(* PLC project TC3_TE1400_GeneratedModule_controller_ballcatcher_FB, Beckhoff Automation GmbH & Co. KG TwinCAT 3 Function - TE1400 1.2.1237 *)
(* stored: companyURL www.beckhoff.com, creationDateTime 2020-10-13T20:18:50 *)

TYPE E_TcMatSimDataAreaType : (NotSpecified := 0, Standard, InputSrc, InputDst, OutputSrc, OutputDst, InternalDa, MArea, RetainDa);
END_TYPE

TYPE ST_TcMatSimObjectDataAreaInfo : STRUCT
  pPlcVar : PVOID;
  pModuleProcImg : PVOID;
  nSize : UDINT;
  nDataAreaId : UDINT;
  eDataAreaType : E_TcMatSimDataAreaType;
END_STRUCT;
END_TYPE

{attribute 'pack_mode' := '4'}
TYPE ST_controller_ballcatcherInitData : STRUCT
  Header : TComInitDataHdr;
  CallByHdr : TComInitDataElmHdr;
  CallBy : TctModuleCallByType;
  ExecutionSequenceHdr : TComInitDataElmHdr;
  ExecutionSequence : TctModuleExecutionSequenceType;
  StepSizeHdr : TComInitDataElmHdr;
  StepSize : TctStepSizeType;
  ExtModeParametersHdr : TComInitDataElmHdr;
  ExtModeParameters : TctExtModeParametersType;
  ExecuteModelCodeHdr : TComInitDataElmHdr;
  ExecuteModelCode : BOOL;
  ModelParametersHdr : TComInitDataElmHdr;
  ModelParameters : P_controller_ballcatcher_T;
  ContextInfoArr_0_TaskOidHdr : TComInitDataElmHdr;
  ContextInfoArr_0_TaskOid : OTCID;
  ContextInfoArr_0_TaskPriorityHdr : TComInitDataElmHdr;
  ContextInfoArr_0_TaskPriority : UDINT;
  ContextInfoArr_0_TaskCycleTimeNsHdr : TComInitDataElmHdr;
  ContextInfoArr_0_TaskCycleTimeNs : UDINT;
  ContextInfoArr_0_TaskPortHdr : TComInitDataElmHdr;
  ContextInfoArr_0_TaskPort : UINT;
  ContextInfoArr_0_TaskSortOrderHdr : TComInitDataElmHdr;
  ContextInfoArr_0_TaskSortOrder : UDINT;
END_STRUCT;
END_TYPE

TYPE ST_controller_ballcatcher_Input : STRUCT
  fast_sensor_torque : matrix_7_real_T;
  fast_sensor_position : matrix_7_real_T;
  fast_sensor_motor_torque_feedback : matrix_7_real_T;
  motion_enabled : LREAL;
  sensor_mft_application_button : LREAL;
  q_d_in : matrix_7_real_T;
  traj_time_interval : matrix_2_real_T;
  traj_update_index : LREAL;
  traj_reset : LREAL;
  chart_state : LREAL;
  controller_select : UDINT;
END_STRUCT;
END_TYPE

TYPE ST_controller_ballcatcher_Output : STRUCT
  fast_control_motor_torque : matrix_7_real_T;
  fast_control_motor_enable : matrix_7_real_T;
  motion_enabled_out : LREAL;
  traj_gen_error : BOOL;
  q_d : matrix_7_real_T;
  q_p_d : matrix_7_real_T;
  q_pp_d : matrix_7_real_T;
END_STRUCT;
END_TYPE

FUNCTION_BLOCK FB_TcMatSimObject
  VAR_INPUT
    bWriteFbInputValues : BOOL := TRUE;  (* set this flag to write FB input values to the TcComObject's input DataAreas. This will overwrite the mapped input values before module execution. Set to FALSE to read the mapped input values from the TcComObject to the FB. *)
  END_VAR
  VAR
    pDataAreas : POINTER TO ST_TcMatSimObjectDataAreaInfo;  (* process image src and dst pointers and sizes *)
    nDataAreas : UDINT;
    ipObjSrv : ITComObjectServer;  (* global interface pointers *)
    ipTcComObj : ITComObject;  (* object interface pointers *)
    ipTcCyclic : ITcCyclic;
    ipTcPostCyclic : ITcPostCyclic;
    ipTcAdi : ITcADI;
    ipTask : ITcTask;  (* task interface pointers *)
    pInitData : POINTER TO TComInitDataHdr;  (* initial parameters *)
    hResult : HRESULT;  (* hResult of interface calls (0 if no error) *)
    moduleClsId : CLSID;  (* module class ID *)
    assignedClsId : CLSID;  (* expected/desired module class ID *)
    bClassIdVerified : BOOL;
    bDynInstance : BOOL;  (* flag indicating whether the module instance was created dynamically *)
    eInitialObjState : TCOM_STATE := TCOM_STATE.TCOM_STATE_INIT;  (* the object state at the time FB_init was called, FB_exit will try to switch to this state (only if this means to shift down) *)
  END_VAR

            
          

{attribute 'object_name' := 'ReleaseTcComInterface'}
METHOD ReleaseTcComInterface : HRESULT
  VAR
    nStateChangeCnt : DINT := 0;
  END_VAR
                  
IF (ipTcComObj<>0) THEN
  WHILE (State>eInitialObjState AND nStateChangeCnt<1000) DO
    State := eInitialObjState;
    nStateChangeCnt := nStateChangeCnt+1;
  END_WHILE
  ReleaseObjInterfaces();
  IF (bDynInstance) THEN
    ReleaseTcComInterface := TC3_MODULE.FW_ObjMgr_DeleteInstance(ADR(ipTcComObj));
  ELSE
    ipTcComObj.TcRelease();
  END_IF
  ipTcComObj := 0;
END_IF
                  
                
END_METHOD

{attribute 'object_name' := 'ReleaseObjInterfaces'}
METHOD ReleaseObjInterfaces : HRESULT
                  
// release interface pointers
IF (ipTcCyclic<>0) THEN
  ipTcCyclic.TcRelease();
  ipTcCyclic := 0;
END_IF
IF (ipTcPostCyclic<>0) THEN
  ipTcPostCyclic.TcRelease();
  ipTcPostCyclic := 0;
END_IF
IF (ipTcAdi<>0) THEN
  ipTcAdi.TcRelease();
  ipTcAdi := 0;
END_IF
                  
                
END_METHOD

{attribute 'object_name' := 'Internal_SetObjState'}
METHOD Internal_SetObjState
  VAR_INPUT
    hr : REFERENCE TO HRESULT;
    nextState : TCOM_STATE;
  END_VAR
                  
// verify class id
IF (SUCCEEDED(hr)) THEN
  hr := VerifyClassId();
END_IF

// switch object state
IF (SUCCEEDED(hr) AND nextState>=TCOM_STATE_INIT) THEN
  IF (ipTcComObj=0) THEN
    hr := Tc2_System.E_HRESULTAdsErr.NOINTERFACE;
  END_IF
  IF (ipObjSrv=0) THEN
    hr := Tc2_System.E_HRESULTAdsErr.NOINTERFACE;
  END_IF
  IF (SUCCEEDED(hr)) THEN
    hr := ipTcComObj.TcSetObjState(nextState,ipObjSrv,pInitData);
  END_IF
END_IF
                  
                
END_METHOD

{attribute 'object_name' := 'FB_init'}
METHOD FB_init : BOOL
  VAR_INPUT
    bInitRetains : BOOL;  (* init retain variables *)
    bInCopyCode : BOOL;  (* Online Change *)
    oid : OTCID;
  END_VAR
                  
FB_init := SUCCEEDED(Init(oid));
                  
                
END_METHOD

{attribute 'object_name' := 'GetObjPara'}
METHOD GetObjPara : HRESULT
  VAR_INPUT
    pid : PTCID;
    nData : UDINT;
    pData : PVOID;
  END_VAR
                  
IF (ipTcComObj=0) THEN
  GetObjPara := Tc2_System.E_HRESULTAdsErr.NOINTERFACE;
END_IF

IF (SUCCEEDED(GetObjPara)) THEN
  GetObjPara := ipTcComObj.TcGetObjPara(pid:=pid,nData,pData,0);
END_IF
                  
                
END_METHOD

{attribute 'object_name' := 'QueryObjInterface'}
METHOD QueryObjInterface
  VAR_INPUT
    hr : REFERENCE TO HRESULT;
    iid : REFERENCE TO IID;
    pipItf : POINTER TO ITcUnknown;
  END_VAR
  VAR CONSTANT
    pNull : PVOID := 0;
  END_VAR
                  
IF (SUCCEEDED(hr)) THEN
  IF (ipTcComObj=0) THEN
    hr := Tc2_System.E_HRESULTAdsErr.NOINTERFACE;
  ELSIF (pipItf^=ULINT_TO_DWORD(pNull)) THEN
    hr := ipTcComObj.TcQueryInterface(iid:= iid, pipItf:=pipItf);
  END_IF
END_IF
                  
                
END_METHOD

{attribute 'object_name' := 'SaveOnlineParametersForInit'}
METHOD SaveOnlineParametersForInit : HRESULT
  VAR
    idx : UINT;
    pInitElemHdr : POINTER TO TComInitDataElmHdr;
    pData : PVOID;
    nData : UDINT;
  END_VAR
  VAR CONSTANT
    nInitDataAlignment : UDINT := 4;
  END_VAR
                  IF (pInitData<>0) THEN
  pInitElemHdr := pInitData + SIZEOF(pInitData^);
  FOR idx:=1 TO pInitData^.uiElmCnt DO
    pData := pInitElemHdr + ULINT_TO_DWORD(SIZEOF(pInitElemHdr^));
    nData := pInitElemHdr^.cbData;
    SaveOnlineParametersForInit := GetObjPara(pInitElemHdr^.indexOffset,nData,pData);
    IF (FAILED(SaveOnlineParametersForInit)) THEN
      RETURN;
    END_IF
    pInitElemHdr := pData + (nInitDataAlignment*((nData + nInitDataAlignment - 1)/nInitDataAlignment));
  END_FOR
ELSE
	SaveOnlineParametersForInit := Tc2_System.E_HRESULTAdsErr.NOTINIT;
END_IF
                  
                
END_METHOD

{attribute 'object_name' := 'ResetHresult'}
METHOD ResetHresult
                  hResult := S_OK;
                
END_METHOD

{attribute 'object_name' := 'Execute'}
METHOD Execute : HRESULT
  VAR
    nDaIdx : UDINT;
    pCurDataArea : POINTER TO ST_TcMatSimObjectDataAreaInfo;
  END_VAR
                  
IF (SUCCEEDED(hResult)) THEN
  hResult := VerifyClassId();
END_IF

IF (SUCCEEDED(hResult) AND State<>TCOM_STATE_OP) THEN
  hResult := Tc2_System.E_HRESULTAdsErr.NOTREADY;
END_IF

// get image pointers
IF (SUCCEEDED(hResult)) THEN
  GetImagePtrs(hResult);
END_IF

// copy inputs
IF (pDataAreas<>0 AND nDataAreas>0 AND bWriteFbInputValues) THEN
  FOR nDaIdx:=0 TO nDataAreas-1 DO
    IF (FAILED(hResult))THEN
      CONTINUE;
    END_IF
    pCurDataArea := pDataAreas + nDaIdx*SIZEOF(ST_TcMatSimObjectDataAreaInfo);
    IF ((pCurDataArea^.eDataAreaType <> E_TcMatSimDataAreaType.InputDst))THEN
      CONTINUE;
    END_IF
    IF (pCurDataArea^.pModuleProcImg<>0 AND pCurDataArea^.pPlcVar<>0) THEN
      MEMCPY(pCurDataArea^.pModuleProcImg,pCurDataArea^.pPlcVar,pCurDataArea^.nSize);
    ELSE
      hResult := Tc2_System.E_HRESULTAdsErr.NOINTERFACE;
    END_IF
  END_FOR
END_IF

// call cycle update
IF (SUCCEEDED(hResult)) THEN
  IF (ipTcCyclic<>0) THEN
    hResult := ipTcCyclic.CycleUpdate(ipTask:= ipTask, ipCaller:= 0, context:= 0);
  ELSE
    hResult := Tc2_System.E_HRESULTAdsErr.NOINTERFACE;
  END_IF
END_IF

// copy outputs
IF (pDataAreas<>0 AND nDataAreas>0) THEN
  FOR nDaIdx:=0 TO nDataAreas-1 DO
    IF (FAILED(hResult))THEN
      CONTINUE;
    END_IF
    pCurDataArea := pDataAreas + nDaIdx*SIZEOF(ST_TcMatSimObjectDataAreaInfo);
    IF ((pCurDataArea^.eDataAreaType = E_TcMatSimDataAreaType.OutputSrc) OR NOT bWriteFbInputValues) THEN
      IF (pCurDataArea^.pModuleProcImg<>0 AND pCurDataArea^.pPlcVar<>0) THEN
        MEMCPY(pCurDataArea^.pPlcVar,pCurDataArea^.pModuleProcImg,pCurDataArea^.nSize);
      ELSE
        hResult := Tc2_System.E_HRESULTAdsErr.NOINTERFACE;
      END_IF
    END_IF
  END_FOR
END_IF


// call post cyclic update
IF (SUCCEEDED(hResult)) THEN
  IF (ipTcPostCyclic<>0) THEN
    hResult := ipTcPostCyclic.PostCyclicUpdate(ipTask:= 0, ipCaller:= 0, context:= 0);
  ELSE
    hResult := Tc2_System.E_HRESULTAdsErr.NOINTERFACE;
  END_IF
END_IF

ReleaseImagePtrs();

Execute := hResult;
                  
                
END_METHOD

{attribute 'object_name' := 'GetImagePtrs'}
METHOD GetImagePtrs
  VAR_INPUT
    hr : REFERENCE TO HRESULT;
  END_VAR
  VAR
    nDaIdx : UDINT;
    pCurDataArea : POINTER TO ST_TcMatSimObjectDataAreaInfo;
  END_VAR
                  
IF (ipTcAdi=0) THEN
  hr := Tc2_System.E_HRESULTAdsErr.NOINTERFACE;
END_IF
IF(State<>TCOM_STATE_OP)THEN
  hr := Tc2_System.E_HRESULTAdsErr.INVALIDSTATE;
END_IF


// get pointers to process images
IF (pDataAreas<>0 AND nDataAreas>0) THEN
  FOR nDaIdx:=0 TO nDataAreas-1 DO
    pCurDataArea := pDataAreas + nDaIdx*SIZEOF(ST_TcMatSimObjectDataAreaInfo);
    IF (FAILED(hr))THEN
      CONTINUE;
    END_IF
    IF ((pCurDataArea^.eDataAreaType <> E_TcMatSimDataAreaType.InputDst) AND (pCurDataArea^.eDataAreaType <> E_TcMatSimDataAreaType.OutputSrc))THEN
      CONTINUE;
    END_IF
    IF (pCurDataArea^.pModuleProcImg=0 AND pCurDataArea^.nSize>0) THEN
      hr := ipTcAdi.GetImagePtr(size:= pCurDataArea^.nSize , offs:=0 , adi_x:=pCurDataArea^.nDataAreaId , ppData:=ADR(pCurDataArea^.pModuleProcImg));
    END_IF
  END_FOR
END_IF

IF (FAILED(hr)) THEN
  ReleaseImagePtrs();
END_IF
                  
                
END_METHOD

{attribute 'object_name' := 'VerifyClassId'}
METHOD VerifyClassId : HRESULT
  VAR
    emptyClsId : CLSID;
  END_VAR
                  memset(ADR(emptyClsId),0,SIZEOF(emptyClsId));
IF (bClassIdVerified) THEN
  // class ID was already verified
  VerifyClassId := Tc2_System.E_HRESULTAdsErr.HRESULT_ADS_NOERROR;
ELSIF (memcmp(ADR(assignedClsId),ADR(emptyClsId),SIZEOF(assignedClsId))=0) THEN
  // skip class ID verification if no assignedClsId specified
  VerifyClassId := Tc2_System.E_HRESULTAdsErr.HRESULT_ADS_NOERROR;
ELSE
  // verify class ID
  VerifyClassId := ReadModuleClassId();

  IF (SUCCEEDED(VerifyClassId)) THEN
    IF (memcmp(ADR(assignedClsId),ADR(moduleClsId),SIZEOF(assignedClsId))<>0) THEN
     VerifyClassId := Tc2_System.E_HRESULTAdsErr.INVALIDCLSID;
    END_IF
  END_IF
  bClassIdVerified := SUCCEEDED(VerifyClassId);
END_IF
                  
                
END_METHOD

{attribute 'object_name' := 'SetObjPara'}
METHOD SetObjPara : HRESULT
  VAR_INPUT
    pid : PTCID;
    nData : UDINT;
    pData : PVOID;
  END_VAR
                  
IF (ipTcComObj=0) THEN
  SetObjPara := Tc2_System.E_HRESULTAdsErr.NOINTERFACE;
END_IF

IF (SUCCEEDED(SetObjPara)) THEN
  SetObjPara := ipTcComObj.TcSetObjPara(pid:=pid,nData,pData,0);
END_IF
                  
                
END_METHOD

{attribute 'object_name' := 'QueryTcComInterface'}
METHOD QueryTcComInterface
  VAR_INPUT
    hr : REFERENCE TO HRESULT;
    oid : OTCID;
  END_VAR
                  
IF (ipObjSrv=0) THEN
  hr := Tc2_System.E_HRESULTAdsErr.NOINTERFACE;
END_IF

IF (SUCCEEDED(hr) AND ipTcComObj=0) THEN
  bDynInstance := FALSE;
  IF(oid>0) THEN
    // query interface of existing object
    hr := ipObjSrv.TcQueryObjectInterface(oid,IID_ITComObject,ADR(ipTcComObj));
  ELSE
    // create new instance and get the object interface
    hr := ipObjSrv.TcCreateInstance(assignedClsId,IID_ITComObject,ADR(ipTcComObj));
    IF (SUCCEEDED(hr)) THEN
      bDynInstance := TRUE;
      hr := ipTcComObj.TcSetObjectId(OTCID_CreateNewId);
    END_IF
  END_IF
  IF (SUCCEEDED(hr)) THEN
    eInitialObjState := State;
  END_IF
END_IF
                  
                
END_METHOD

{attribute 'object_name' := 'ReleaseImagePtrs'}
METHOD ReleaseImagePtrs : HRESULT
  VAR
    nDaIdx : UDINT;
    pCurDataArea : POINTER TO ST_TcMatSimObjectDataAreaInfo;
  END_VAR
                  
IF (ipTcAdi=0) THEN
  ReleaseImagePtrs := Tc2_System.E_HRESULTAdsErr.NOINTERFACE;
END_IF

IF (SUCCEEDED(ReleaseImagePtrs) AND pDataAreas<>0 AND nDataAreas>0) THEN
  // release pointers to the simulink module process images
  FOR nDaIdx:=0 TO nDataAreas-1 DO
    pCurDataArea := pDataAreas + nDaIdx*SIZEOF(ST_TcMatSimObjectDataAreaInfo);

    IF (pCurDataArea^.pModuleProcImg<>0) THEN
      ipTcAdi.ReleaseImagePtr(pData:=pCurDataArea^.pModuleProcImg);
      pCurDataArea^.pModuleProcImg := 0;
    END_IF
  END_FOR
END_IF
                  
                
END_METHOD

{attribute 'object_name' := 'FB_exit'}
METHOD FB_exit : BOOL
  VAR_INPUT
    bInCopyCode : BOOL;  (* Online Change *)
  END_VAR
                  
IF (NOT bInCopyCode) THEN
  IF (ipObjSrv<>0) THEN
    ipObjSrv.TcRelease();
    ipObjSrv := 0;
  END_IF

  ReleaseTcComInterface();
END_IF
                  
                
END_METHOD

{attribute 'object_name' := 'InitObjName'}
METHOD InitObjName
  VAR_INPUT
    hr : REFERENCE TO HRESULT;
  END_VAR
  VAR
    objectName : STRING(255) := 'TcMatSimObject_PlcRtFbInstance';
    oid : OTCID;
  END_VAR
                  
IF (SUCCEEDED(hr)) THEN
  hr := ipTcComObj.TcGetObjectId(oid);
END_IF

IF (SUCCEEDED(hr) and bDynInstance) THEN
  objectName := TC2_STANDARD.CONCAT(objectName,'_');
  objectName := TC2_STANDARD.CONCAT(objectName,UDINT_TO_STRING(oid));
  hr := ipTcComObj.TcSetObjectName(ADR(objectName));
END_IF
                  
                
END_METHOD

{attribute 'object_name' := 'SetObjState'}
METHOD SetObjState : HRESULT
  VAR_INPUT
    finalState : TCOM_STATE;
  END_VAR
  VAR
    bShiftUp : BOOL;
    bShiftDown : BOOL;
    currentState : TCOM_STATE;
  END_VAR
                  
currentState := State;

bShiftUp := finalState>currentState;
bShiftDown := finalState<currentState;

// do not switch up on error
IF (FAILED(hresult)) THEN
  bShiftUp := FALSE;
END_IF
// reset existing error on switching down
IF (bShiftDown) THEN
  ResetHresult();
END_IF

// prepared state switch
CASE currentState OF
  TCOM_STATE_INIT:
    IF(bShiftUp) THEN
      QueryTcComInterface(hResult,0);
      Internal_SetObjState(hResult,TCOM_STATE.TCOM_STATE_PREOP);
      InitObjName(hResult);
    END_IF

  TCOM_STATE_PREOP:
    IF(bShiftUp) THEN
      Internal_SetObjState(hResult,TCOM_STATE.TCOM_STATE_SAFEOP);
      QueryObjInterfaces(hResult);
    ELSIF (bShiftDown) THEN
      Internal_SetObjState(hResult,TCOM_STATE.TCOM_STATE_INIT);
    END_IF

  TCOM_STATE_SAFEOP:
    IF(bShiftUp) THEN
      Internal_SetObjState(hResult,TCOM_STATE.TCOM_STATE_OP);
      QueryObjInterfaces(hResult);
    ELSIF (bShiftDown) THEN
      Internal_SetObjState(hResult,TCOM_STATE.TCOM_STATE_PREOP);
      ReleaseObjInterfaces();
    END_IF


  TCOM_STATE_OP:
    IF (bShiftDown) THEN
      Internal_SetObjState(hResult,TCOM_STATE.TCOM_STATE_SAFEOP);
    END_IF
END_CASE

SetObjState := hResult;
                  
                
END_METHOD

{attribute 'object_name' := 'QueryObjInterfaces'}
METHOD QueryObjInterfaces
  VAR_INPUT
    hr : REFERENCE TO HRESULT;
  END_VAR
                  
IF(State<TCOM_STATE_PREOP)THEN
  hr := Tc2_System.E_HRESULTAdsErr.INVALIDSTATE;
END_IF

//cyclic interface
QueryObjInterface(hr,IID_ITCCYCLIC,ADR(ipTcCyclic));
//post cyclic interface
QueryObjInterface(hr,IID_ITCPOSTCYCLIC,ADR(ipTcPostCyclic));
//adi interface
QueryObjInterface(hr,IID_ITcADI,ADR(ipTcAdi));
                  
                
END_METHOD

{attribute 'object_name' := 'Init'}
METHOD Init : HRESULT
  VAR_INPUT
    oid : OTCID;
  END_VAR
                  
// preinitialize variables
memset(ADR(moduleClsId),0,SIZEOF(moduleClsId));
bClassIdVerified := FALSE;
hResult := Tc2_System.E_HRESULTAdsErr.HRESULT_ADS_NOERROR;

// get object server
IF (ipObjSrv=0) THEN
  hResult := FW_ObjMgr_GetObjectServer(_AppInfo.ObjId,ADR(ipObjSrv));
END_IF

// try to get object interfaces
IF (SUCCEEDED(hresult)) THEN
  QueryTcComInterface(hResult,oid);
END_IF

// verify class id
IF (SUCCEEDED(hresult)) THEN
  hresult := VerifyClassId();
END_IF

// query interfaces, if the current state is higher than INIT
IF (SUCCEEDED(hresult) AND State>TCOM_STATE.TCOM_STATE_INIT) THEN
  QueryObjInterfaces(hResult);
END_IF

// return value
Init := hresult;
                  
                
END_METHOD

{attribute 'object_name' := 'ReadModuleClassId'}
METHOD ReadModuleClassId : HRESULT
  VAR
    emptyClsId : CLSID;
  END_VAR
                  memset(ADR(emptyClsId),0,SIZEOF(emptyClsId));
IF (memcmp(ADR(moduleClsId),ADR(emptyClsId),SIZEOF(moduleClsId))=0) THEN
  IF (ipTcComObj=0) THEN
    ReadModuleClassId := Tc2_System.E_HRESULTAdsErr.NOINTERFACE;
  END_IF

  //objectClsId := clsid;
  IF (SUCCEEDED(ReadModuleClassId)) THEN
    ReadModuleClassId := ipTcComObj.GetClassId(moduleClsId);
  END_IF
END_IF
                
END_METHOD

METHOD PUBLIC AssignClassId
VAR_INPUT
	clsId : CLSID;
END_VAR
                  assignedClsId := clsId;
bClassIdVerified := false;
                  
                
END_METHOD

PROPERTY Error : BOOL
GET
                    Error := FAILED(hResult);
                  
END_GET
END_PROPERTY

METHOD PUBLIC SetDataAreaInfo
VAR_INPUT
  pDataAreas: POINTER TO ST_TcMatSimObjectDataAreaInfo;
  nDataAreas: UDINT;
END_VAR
                  
THIS^.nDataAreas := nDataAreas;
THIS^.pDataAreas := pDataAreas;
                  
                
END_METHOD

METHOD PUBLIC SetInitDataInfo
VAR_INPUT
  pInitData : POINTER TO TComInitDataHdr;
END_VAR
                  this^.pInitData := pInitData;
                
END_METHOD

PROPERTY ClassId : CLSID
GET
                    hResult := ReadModuleClassId();
ClassId := moduleClsId;
                    
                  
END_GET
END_PROPERTY

PROPERTY State : TCOM_STATE
GET
  VAR
    hr : HRESULT := S_OK;
    eObjState : TCOM_STATE;
  END_VAR
                    
IF (ipTcComObj<>0) THEN
  hr := ipTcComObj.TcGetObjState(ADR(eObjState));
IF (FAILED(hr)) THEN
  eObjState := TCOM_STATE.TCOM_STATE_INIT;
END_IF
ELSE
  eObjState := TCOM_STATE.TCOM_STATE_INIT;
END_IF
State := eObjState;
                    
                  
END_GET
SET
                    SetObjState(State);
                  
END_SET
END_PROPERTY

PROPERTY ErrorCode : HRESULT
GET
                    ErrorCode := hResult;
                  
END_GET
END_PROPERTY
END_FUNCTION_BLOCK

{attribute 'TcDependOnClassFactory' := 'controller_ballcatcher'}
FUNCTION_BLOCK FB_controller_ballcatcher EXTENDS FB_TcMatSimObject
  VAR_INPUT
    stInput : ST_controller_ballcatcher_Input;
  END_VAR
  VAR_OUTPUT
    stOutput : ST_controller_ballcatcher_Output;
  END_VAR
  VAR
    stInitData : ST_controller_ballcatcherInitData;
    arrDataAreas : ARRAY[1..2] OF ST_TcMatSimObjectDataAreaInfo;
    bParametersVerified : BOOL;
  END_VAR

            
          

{attribute 'object_name' := 'Internal_SetObjState'}
METHOD Internal_SetObjState
  VAR_INPUT
    hr : REFERENCE TO HRESULT;
    nextState : TCOM_STATE;
  END_VAR
                  
// update pointer to InitData structure
SetInitDataInfo(ADR(stInitData));
// call base method
SUPER^.Internal_SetObjState(hr,nextState);
                  
                
END_METHOD

{attribute 'object_name' := 'SaveOnlineParametersForInit'}
METHOD SaveOnlineParametersForInit : HRESULT
  VAR
    idx : UINT;
    pInitElemHdr : POINTER TO TComInitDataElmHdr;
    pData : PVOID;
    nData : UDINT;
  END_VAR
  VAR CONSTANT
    nInitDataAlignment : UDINT := 4;
  END_VAR
                  
// update pointer to InitData structure
SetInitDataInfo(ADR(stInitData));
// call base method
SaveOnlineParametersForInit := SUPER^.SaveOnlineParametersForInit();
                  
                
END_METHOD

METHOD FB_init : BOOL
  VAR_INPUT
    bInitRetains : BOOL;  (* if TRUE, the retain variables are initialized (warm start / cold start) *)
    bInCopyCode : BOOL;  (* if TRUE, the instance afterwards gets moved into the copy code (online change) *)
    oid : OTCID;
  END_VAR
  VAR
    clsId : CLSID;
  END_VAR
                  
// initialize flags
bParametersVerified := false;
                    
// set module class id for compatibility check
clsId.Data1 := 16#fc150844;
clsId.Data2 := 16#4666;
clsId.Data3 := 16#4420;
clsId.Data4[0] := 16#8f;
clsId.Data4[1] := 16#db;
clsId.Data4[2] := 16#90;
clsId.Data4[3] := 16#b5;
clsId.Data4[4] := 16#fc;
clsId.Data4[5] := 16#68;
clsId.Data4[6] := 16#4e;
clsId.Data4[7] := 16#ee;

AssignClassId(clsId);
                    
// initialize InitData structure with default values              
stInitData.CallByHdr.indexGroup := 0;
stInitData.CallByHdr.indexOffset := 16#00000000;
stInitData.CallByHdr.cbData := SIZEOF(stInitData.CallBy);
stInitData.CallBy := TctModuleCallByType.CyclicTask;
stInitData.ExecutionSequenceHdr.indexGroup := 0;
stInitData.ExecutionSequenceHdr.indexOffset := 16#00000001;
stInitData.ExecutionSequenceHdr.cbData := SIZEOF(stInitData.ExecutionSequence);
stInitData.ExecutionSequence := TctModuleExecutionSequenceType.StateUpdateAfterOutputMapping;
stInitData.StepSizeHdr.indexGroup := 0;
stInitData.StepSizeHdr.indexOffset := 16#00000002;
stInitData.StepSizeHdr.cbData := SIZEOF(stInitData.StepSize);
stInitData.StepSize := TctStepSizeType.RequireMatchingTaskCycleTime;
stInitData.ExtModeParametersHdr.indexGroup := 0;
stInitData.ExtModeParametersHdr.indexOffset := 16#bf002000;
stInitData.ExtModeParametersHdr.cbData := SIZEOF(stInitData.ExtModeParameters);
stInitData.ExtModeParameters.ConnectionTimeout := 3;
stInitData.ExtModeParameters.InitIncomingPktBufferSize := 10000;
stInitData.ExtModeParameters.InitOutgoingPktBufferSize := 10000;
stInitData.ExtModeParameters.Activated := 1;
stInitData.ExtModeParameters.AllowExecutionCommands := 1;
stInitData.ExtModeParameters.WaitForStartCommand := 0;
stInitData.ExtModeParameters.AllowParameterChange := 1;
stInitData.ExecuteModelCodeHdr.indexGroup := 0;
stInitData.ExecuteModelCodeHdr.indexOffset := 16#00000008;
stInitData.ExecuteModelCodeHdr.cbData := SIZEOF(stInitData.ExecuteModelCode);
stInitData.ExecuteModelCode := 1;
stInitData.ModelParametersHdr.indexGroup := 0;
stInitData.ModelParametersHdr.indexOffset := 16#83000000;
stInitData.ModelParametersHdr.cbData := SIZEOF(stInitData.ModelParameters);
stInitData.ModelParameters.param_robot.hanging := 0;
stInitData.ModelParameters.param_robot.R_0[0] := 1;
stInitData.ModelParameters.param_robot.R_0[1] := 0;
stInitData.ModelParameters.param_robot.R_0[2] := 0;
stInitData.ModelParameters.param_robot.R_0[3] := 0;
stInitData.ModelParameters.param_robot.R_0[4] := 1;
stInitData.ModelParameters.param_robot.R_0[5] := 0;
stInitData.ModelParameters.param_robot.R_0[6] := 0;
stInitData.ModelParameters.param_robot.R_0[7] := 0;
stInitData.ModelParameters.param_robot.R_0[8] := 1;
stInitData.ModelParameters.param_robot.p_0[0] := 0;
stInitData.ModelParameters.param_robot.p_0[1] := 0;
stInitData.ModelParameters.param_robot.p_0[2] := 0;
stInitData.ModelParameters.param_robot.n := 7;
stInitData.ModelParameters.param_robot.g := 9.8100000000000005;
stInitData.ModelParameters.param_robot.beta := 0;
stInitData.ModelParameters.param_robot.l_0 := 0.1525;
stInitData.ModelParameters.param_robot.l_1 := 0.20749999999999999;
stInitData.ModelParameters.param_robot.l_2 := 0.23250000000000001;
stInitData.ModelParameters.param_robot.l_3 := 0.1875;
stInitData.ModelParameters.param_robot.l_4 := 0.21249999999999999;
stInitData.ModelParameters.param_robot.l_5 := 0.1875;
stInitData.ModelParameters.param_robot.l_6 := 0.079600000000000004;
stInitData.ModelParameters.param_robot.l_7 := 0.072400000000000006;
stInitData.ModelParameters.param_robot.d_1 := 0.012999999999999999;
stInitData.ModelParameters.param_robot.d_3 := 0.010999999999999999;
stInitData.ModelParameters.param_robot.d_5 := 0.062;
stInitData.ModelParameters.param_robot.m_l1 := 6.4950000000000001;
stInitData.ModelParameters.param_robot.m_l2 := 8.8070000000000004;
stInitData.ModelParameters.param_robot.m_l3 := 2.7999999999999998;
stInitData.ModelParameters.param_robot.m_l4 := 5.2830000000000004;
stInitData.ModelParameters.param_robot.m_l5 := 1.889;
stInitData.ModelParameters.param_robot.m_l6 := 2.3199999999999998;
stInitData.ModelParameters.param_robot.m_l7 := 0.86299999999999999;
stInitData.ModelParameters.param_robot.s_l1x := 0;
stInitData.ModelParameters.param_robot.s_l1y := -0.01439;
stInitData.ModelParameters.param_robot.s_l1z := 0.102503;
stInitData.ModelParameters.param_robot.s_l2x := -1.2e-05;
stInitData.ModelParameters.param_robot.s_l2y := -0.06472;
stInitData.ModelParameters.param_robot.s_l2z := 0.017804;
stInitData.ModelParameters.param_robot.s_l3x := -0.00020799999999999999;
stInitData.ModelParameters.param_robot.s_l3y := 0.01601;
stInitData.ModelParameters.param_robot.s_l3z := 0.087282999999999999;
stInitData.ModelParameters.param_robot.s_l4x := -0.000203;
stInitData.ModelParameters.param_robot.s_l4y := 0.098639000000000004;
stInitData.ModelParameters.param_robot.s_l4z := 0.022478000000000001;
stInitData.ModelParameters.param_robot.s_l5x := -5.7000000000000003e-05;
stInitData.ModelParameters.param_robot.s_l5y := -0.014468;
stInitData.ModelParameters.param_robot.s_l5z := 0.062937999999999994;
stInitData.ModelParameters.param_robot.s_l6x := -0.00036299999999999999;
stInitData.ModelParameters.param_robot.s_l6y := -0.016982000000000001;
stInitData.ModelParameters.param_robot.s_l6z := 0.042269000000000001;
stInitData.ModelParameters.param_robot.s_l7x := 0.0019040000000000003;
stInitData.ModelParameters.param_robot.s_l7y := -9.2999999999999997e-05;
stInitData.ModelParameters.param_robot.s_l7z := 0.018862000000000004;
stInitData.ModelParameters.param_robot.I_l1xx := 0.0690761441316632;
stInitData.ModelParameters.param_robot.I_l1yy := 0.071108558691451398;
stInitData.ModelParameters.param_robot.I_l1zz := 0.020062585440211899;
stInitData.ModelParameters.param_robot.I_l2xx := 0.082470168353469195;
stInitData.ModelParameters.param_robot.I_l2yy := 0.016411096805519099;
stInitData.ModelParameters.param_robot.I_l2zz := 0.087351089266136106;
stInitData.ModelParameters.param_robot.I_l3xx := 0.023015294131881699;
stInitData.ModelParameters.param_robot.I_l3yy := 0.022866155414347399;
stInitData.ModelParameters.param_robot.I_l3zz := 0.055448228374898302;
stInitData.ModelParameters.param_robot.I_l4xx := 0.047278966834196801;
stInitData.ModelParameters.param_robot.I_l4yy := 0.0096472680414690908;
stInitData.ModelParameters.param_robot.I_l4zz := 0.046652900776167898;
stInitData.ModelParameters.param_robot.I_l5xx := 0.0138359953358589;
stInitData.ModelParameters.param_robot.I_l5yy := 0.011685933775196901;
stInitData.ModelParameters.param_robot.I_l5zz := 0.00571863785412578;
stInitData.ModelParameters.param_robot.I_l6xx := 0.0073275878721676497;
stInitData.ModelParameters.param_robot.I_l6yy := 0.0047763375578371101;
stInitData.ModelParameters.param_robot.I_l6zz := 0.0060679763855029604;
stInitData.ModelParameters.param_robot.I_l7xx := 0.00088400000000000002;
stInitData.ModelParameters.param_robot.I_l7yy := 0.00088800000000000001;
stInitData.ModelParameters.param_robot.I_l7zz := 0.0011050000000000001;
stInitData.ModelParameters.param_robot.n_1 := 160;
stInitData.ModelParameters.param_robot.n_2 := 160;
stInitData.ModelParameters.param_robot.n_3 := 160;
stInitData.ModelParameters.param_robot.n_4 := 160;
stInitData.ModelParameters.param_robot.n_5 := 100;
stInitData.ModelParameters.param_robot.n_6 := 160;
stInitData.ModelParameters.param_robot.n_7 := 160;
stInitData.ModelParameters.param_robot.N[0] := 160;
stInitData.ModelParameters.param_robot.N[1] := 0;
stInitData.ModelParameters.param_robot.N[2] := 0;
stInitData.ModelParameters.param_robot.N[3] := 0;
stInitData.ModelParameters.param_robot.N[4] := 0;
stInitData.ModelParameters.param_robot.N[5] := 0;
stInitData.ModelParameters.param_robot.N[6] := 0;
stInitData.ModelParameters.param_robot.N[7] := 0;
stInitData.ModelParameters.param_robot.N[8] := 160;
stInitData.ModelParameters.param_robot.N[9] := 0;
stInitData.ModelParameters.param_robot.N[10] := 0;
stInitData.ModelParameters.param_robot.N[11] := 0;
stInitData.ModelParameters.param_robot.N[12] := 0;
stInitData.ModelParameters.param_robot.N[13] := 0;
stInitData.ModelParameters.param_robot.N[14] := 0;
stInitData.ModelParameters.param_robot.N[15] := 0;
stInitData.ModelParameters.param_robot.N[16] := 160;
stInitData.ModelParameters.param_robot.N[17] := 0;
stInitData.ModelParameters.param_robot.N[18] := 0;
stInitData.ModelParameters.param_robot.N[19] := 0;
stInitData.ModelParameters.param_robot.N[20] := 0;
stInitData.ModelParameters.param_robot.N[21] := 0;
stInitData.ModelParameters.param_robot.N[22] := 0;
stInitData.ModelParameters.param_robot.N[23] := 0;
stInitData.ModelParameters.param_robot.N[24] := 160;
stInitData.ModelParameters.param_robot.N[25] := 0;
stInitData.ModelParameters.param_robot.N[26] := 0;
stInitData.ModelParameters.param_robot.N[27] := 0;
stInitData.ModelParameters.param_robot.N[28] := 0;
stInitData.ModelParameters.param_robot.N[29] := 0;
stInitData.ModelParameters.param_robot.N[30] := 0;
stInitData.ModelParameters.param_robot.N[31] := 0;
stInitData.ModelParameters.param_robot.N[32] := 100;
stInitData.ModelParameters.param_robot.N[33] := 0;
stInitData.ModelParameters.param_robot.N[34] := 0;
stInitData.ModelParameters.param_robot.N[35] := 0;
stInitData.ModelParameters.param_robot.N[36] := 0;
stInitData.ModelParameters.param_robot.N[37] := 0;
stInitData.ModelParameters.param_robot.N[38] := 0;
stInitData.ModelParameters.param_robot.N[39] := 0;
stInitData.ModelParameters.param_robot.N[40] := 160;
stInitData.ModelParameters.param_robot.N[41] := 0;
stInitData.ModelParameters.param_robot.N[42] := 0;
stInitData.ModelParameters.param_robot.N[43] := 0;
stInitData.ModelParameters.param_robot.N[44] := 0;
stInitData.ModelParameters.param_robot.N[45] := 0;
stInitData.ModelParameters.param_robot.N[46] := 0;
stInitData.ModelParameters.param_robot.N[47] := 0;
stInitData.ModelParameters.param_robot.N[48] := 160;
stInitData.ModelParameters.param_robot.I_r1xx := 0.000185;
stInitData.ModelParameters.param_robot.I_r1yy := 0.000185;
stInitData.ModelParameters.param_robot.I_r1zz := 0.00042316695312500003;
stInitData.ModelParameters.param_robot.I_r2xx := 0.000185;
stInitData.ModelParameters.param_robot.I_r2yy := 0.000185;
stInitData.ModelParameters.param_robot.I_r2zz := 0.00042316695312500003;
stInitData.ModelParameters.param_robot.I_r3xx := 0.00012899999999999999;
stInitData.ModelParameters.param_robot.I_r3yy := 0.00012899999999999999;
stInitData.ModelParameters.param_robot.I_r3zz := 0.0001910384375;
stInitData.ModelParameters.param_robot.I_r4xx := 0.00012899999999999999;
stInitData.ModelParameters.param_robot.I_r4yy := 0.00012899999999999999;
stInitData.ModelParameters.param_robot.I_r4zz := 0.0001910384375;
stInitData.ModelParameters.param_robot.I_r5xx := 7.4999999999999993e-05;
stInitData.ModelParameters.param_robot.I_r5yy := 7.4999999999999993e-05;
stInitData.ModelParameters.param_robot.I_r5zz := 0.00014709679999999999;
stInitData.ModelParameters.param_robot.I_r6xx := 1.5e-05;
stInitData.ModelParameters.param_robot.I_r6yy := 1.5e-05;
stInitData.ModelParameters.param_robot.I_r6zz := 1.851125e-05;
stInitData.ModelParameters.param_robot.I_r7xx := 1.5e-05;
stInitData.ModelParameters.param_robot.I_r7yy := 1.5e-05;
stInitData.ModelParameters.param_robot.I_r7zz := 1.851125e-05;
stInitData.ModelParameters.param_robot.B[0] := 10.833074000000002;
stInitData.ModelParameters.param_robot.B[1] := 0;
stInitData.ModelParameters.param_robot.B[2] := 0;
stInitData.ModelParameters.param_robot.B[3] := 0;
stInitData.ModelParameters.param_robot.B[4] := 0;
stInitData.ModelParameters.param_robot.B[5] := 0;
stInitData.ModelParameters.param_robot.B[6] := 0;
stInitData.ModelParameters.param_robot.B[7] := 0;
stInitData.ModelParameters.param_robot.B[8] := 10.833074000000002;
stInitData.ModelParameters.param_robot.B[9] := 0;
stInitData.ModelParameters.param_robot.B[10] := 0;
stInitData.ModelParameters.param_robot.B[11] := 0;
stInitData.ModelParameters.param_robot.B[12] := 0;
stInitData.ModelParameters.param_robot.B[13] := 0;
stInitData.ModelParameters.param_robot.B[14] := 0;
stInitData.ModelParameters.param_robot.B[15] := 0;
stInitData.ModelParameters.param_robot.B[16] := 4.8905839999999996;
stInitData.ModelParameters.param_robot.B[17] := 0;
stInitData.ModelParameters.param_robot.B[18] := 0;
stInitData.ModelParameters.param_robot.B[19] := 0;
stInitData.ModelParameters.param_robot.B[20] := 0;
stInitData.ModelParameters.param_robot.B[21] := 0;
stInitData.ModelParameters.param_robot.B[22] := 0;
stInitData.ModelParameters.param_robot.B[23] := 0;
stInitData.ModelParameters.param_robot.B[24] := 4.8905839999999996;
stInitData.ModelParameters.param_robot.B[25] := 0;
stInitData.ModelParameters.param_robot.B[26] := 0;
stInitData.ModelParameters.param_robot.B[27] := 0;
stInitData.ModelParameters.param_robot.B[28] := 0;
stInitData.ModelParameters.param_robot.B[29] := 0;
stInitData.ModelParameters.param_robot.B[30] := 0;
stInitData.ModelParameters.param_robot.B[31] := 0;
stInitData.ModelParameters.param_robot.B[32] := 1.4709679999999998;
stInitData.ModelParameters.param_robot.B[33] := 0;
stInitData.ModelParameters.param_robot.B[34] := 0;
stInitData.ModelParameters.param_robot.B[35] := 0;
stInitData.ModelParameters.param_robot.B[36] := 0;
stInitData.ModelParameters.param_robot.B[37] := 0;
stInitData.ModelParameters.param_robot.B[38] := 0;
stInitData.ModelParameters.param_robot.B[39] := 0;
stInitData.ModelParameters.param_robot.B[40] := 0.47388799999999998;
stInitData.ModelParameters.param_robot.B[41] := 0;
stInitData.ModelParameters.param_robot.B[42] := 0;
stInitData.ModelParameters.param_robot.B[43] := 0;
stInitData.ModelParameters.param_robot.B[44] := 0;
stInitData.ModelParameters.param_robot.B[45] := 0;
stInitData.ModelParameters.param_robot.B[46] := 0;
stInitData.ModelParameters.param_robot.B[47] := 0;
stInitData.ModelParameters.param_robot.B[48] := 0.47388799999999998;
stInitData.ModelParameters.param_robot.K_1 := 60000;
stInitData.ModelParameters.param_robot.K_2 := 60000;
stInitData.ModelParameters.param_robot.K_3 := 40000;
stInitData.ModelParameters.param_robot.K_4 := 40000;
stInitData.ModelParameters.param_robot.K_5 := 40000;
stInitData.ModelParameters.param_robot.K_6 := 20000;
stInitData.ModelParameters.param_robot.K_7 := 20000;
stInitData.ModelParameters.param_robot.K[0] := 60000;
stInitData.ModelParameters.param_robot.K[1] := 0;
stInitData.ModelParameters.param_robot.K[2] := 0;
stInitData.ModelParameters.param_robot.K[3] := 0;
stInitData.ModelParameters.param_robot.K[4] := 0;
stInitData.ModelParameters.param_robot.K[5] := 0;
stInitData.ModelParameters.param_robot.K[6] := 0;
stInitData.ModelParameters.param_robot.K[7] := 0;
stInitData.ModelParameters.param_robot.K[8] := 60000;
stInitData.ModelParameters.param_robot.K[9] := 0;
stInitData.ModelParameters.param_robot.K[10] := 0;
stInitData.ModelParameters.param_robot.K[11] := 0;
stInitData.ModelParameters.param_robot.K[12] := 0;
stInitData.ModelParameters.param_robot.K[13] := 0;
stInitData.ModelParameters.param_robot.K[14] := 0;
stInitData.ModelParameters.param_robot.K[15] := 0;
stInitData.ModelParameters.param_robot.K[16] := 40000;
stInitData.ModelParameters.param_robot.K[17] := 0;
stInitData.ModelParameters.param_robot.K[18] := 0;
stInitData.ModelParameters.param_robot.K[19] := 0;
stInitData.ModelParameters.param_robot.K[20] := 0;
stInitData.ModelParameters.param_robot.K[21] := 0;
stInitData.ModelParameters.param_robot.K[22] := 0;
stInitData.ModelParameters.param_robot.K[23] := 0;
stInitData.ModelParameters.param_robot.K[24] := 40000;
stInitData.ModelParameters.param_robot.K[25] := 0;
stInitData.ModelParameters.param_robot.K[26] := 0;
stInitData.ModelParameters.param_robot.K[27] := 0;
stInitData.ModelParameters.param_robot.K[28] := 0;
stInitData.ModelParameters.param_robot.K[29] := 0;
stInitData.ModelParameters.param_robot.K[30] := 0;
stInitData.ModelParameters.param_robot.K[31] := 0;
stInitData.ModelParameters.param_robot.K[32] := 40000;
stInitData.ModelParameters.param_robot.K[33] := 0;
stInitData.ModelParameters.param_robot.K[34] := 0;
stInitData.ModelParameters.param_robot.K[35] := 0;
stInitData.ModelParameters.param_robot.K[36] := 0;
stInitData.ModelParameters.param_robot.K[37] := 0;
stInitData.ModelParameters.param_robot.K[38] := 0;
stInitData.ModelParameters.param_robot.K[39] := 0;
stInitData.ModelParameters.param_robot.K[40] := 20000;
stInitData.ModelParameters.param_robot.K[41] := 0;
stInitData.ModelParameters.param_robot.K[42] := 0;
stInitData.ModelParameters.param_robot.K[43] := 0;
stInitData.ModelParameters.param_robot.K[44] := 0;
stInitData.ModelParameters.param_robot.K[45] := 0;
stInitData.ModelParameters.param_robot.K[46] := 0;
stInitData.ModelParameters.param_robot.K[47] := 0;
stInitData.ModelParameters.param_robot.K[48] := 20000;
stInitData.ModelParameters.param_robot.tau_max[0] := 320;
stInitData.ModelParameters.param_robot.tau_max[1] := 0;
stInitData.ModelParameters.param_robot.tau_max[2] := 0;
stInitData.ModelParameters.param_robot.tau_max[3] := 0;
stInitData.ModelParameters.param_robot.tau_max[4] := 0;
stInitData.ModelParameters.param_robot.tau_max[5] := 0;
stInitData.ModelParameters.param_robot.tau_max[6] := 0;
stInitData.ModelParameters.param_robot.tau_max[7] := 0;
stInitData.ModelParameters.param_robot.tau_max[8] := 320;
stInitData.ModelParameters.param_robot.tau_max[9] := 0;
stInitData.ModelParameters.param_robot.tau_max[10] := 0;
stInitData.ModelParameters.param_robot.tau_max[11] := 0;
stInitData.ModelParameters.param_robot.tau_max[12] := 0;
stInitData.ModelParameters.param_robot.tau_max[13] := 0;
stInitData.ModelParameters.param_robot.tau_max[14] := 0;
stInitData.ModelParameters.param_robot.tau_max[15] := 0;
stInitData.ModelParameters.param_robot.tau_max[16] := 176;
stInitData.ModelParameters.param_robot.tau_max[17] := 0;
stInitData.ModelParameters.param_robot.tau_max[18] := 0;
stInitData.ModelParameters.param_robot.tau_max[19] := 0;
stInitData.ModelParameters.param_robot.tau_max[20] := 0;
stInitData.ModelParameters.param_robot.tau_max[21] := 0;
stInitData.ModelParameters.param_robot.tau_max[22] := 0;
stInitData.ModelParameters.param_robot.tau_max[23] := 0;
stInitData.ModelParameters.param_robot.tau_max[24] := 176;
stInitData.ModelParameters.param_robot.tau_max[25] := 0;
stInitData.ModelParameters.param_robot.tau_max[26] := 0;
stInitData.ModelParameters.param_robot.tau_max[27] := 0;
stInitData.ModelParameters.param_robot.tau_max[28] := 0;
stInitData.ModelParameters.param_robot.tau_max[29] := 0;
stInitData.ModelParameters.param_robot.tau_max[30] := 0;
stInitData.ModelParameters.param_robot.tau_max[31] := 0;
stInitData.ModelParameters.param_robot.tau_max[32] := 110;
stInitData.ModelParameters.param_robot.tau_max[33] := 0;
stInitData.ModelParameters.param_robot.tau_max[34] := 0;
stInitData.ModelParameters.param_robot.tau_max[35] := 0;
stInitData.ModelParameters.param_robot.tau_max[36] := 0;
stInitData.ModelParameters.param_robot.tau_max[37] := 0;
stInitData.ModelParameters.param_robot.tau_max[38] := 0;
stInitData.ModelParameters.param_robot.tau_max[39] := 0;
stInitData.ModelParameters.param_robot.tau_max[40] := 40;
stInitData.ModelParameters.param_robot.tau_max[41] := 0;
stInitData.ModelParameters.param_robot.tau_max[42] := 0;
stInitData.ModelParameters.param_robot.tau_max[43] := 0;
stInitData.ModelParameters.param_robot.tau_max[44] := 0;
stInitData.ModelParameters.param_robot.tau_max[45] := 0;
stInitData.ModelParameters.param_robot.tau_max[46] := 0;
stInitData.ModelParameters.param_robot.tau_max[47] := 0;
stInitData.ModelParameters.param_robot.tau_max[48] := 40;
stInitData.ModelParameters.param_robot.tau_saturation_max[0] := 160;
stInitData.ModelParameters.param_robot.tau_saturation_max[1] := 160;
stInitData.ModelParameters.param_robot.tau_saturation_max[2] := 88;
stInitData.ModelParameters.param_robot.tau_saturation_max[3] := 88;
stInitData.ModelParameters.param_robot.tau_saturation_max[4] := 55;
stInitData.ModelParameters.param_robot.tau_saturation_max[5] := 20;
stInitData.ModelParameters.param_robot.tau_saturation_max[6] := 20;
stInitData.ModelParameters.param_robot.q_limit_upper[0] := 2.9670597283903604;
stInitData.ModelParameters.param_robot.q_limit_upper[1] := 2.0943951023931953;
stInitData.ModelParameters.param_robot.q_limit_upper[2] := 2.9670597283903604;
stInitData.ModelParameters.param_robot.q_limit_upper[3] := 2.0943951023931953;
stInitData.ModelParameters.param_robot.q_limit_upper[4] := 2.9670597283903604;
stInitData.ModelParameters.param_robot.q_limit_upper[5] := 2.0943951023931953;
stInitData.ModelParameters.param_robot.q_limit_upper[6] := 3.0543261909900763;
stInitData.ModelParameters.param_robot.q_limit_lower[0] := -2.9670597283903604;
stInitData.ModelParameters.param_robot.q_limit_lower[1] := -2.0943951023931953;
stInitData.ModelParameters.param_robot.q_limit_lower[2] := -2.9670597283903604;
stInitData.ModelParameters.param_robot.q_limit_lower[3] := -2.0943951023931953;
stInitData.ModelParameters.param_robot.q_limit_lower[4] := -2.9670597283903604;
stInitData.ModelParameters.param_robot.q_limit_lower[5] := -2.0943951023931953;
stInitData.ModelParameters.param_robot.q_limit_lower[6] := -3.0543261909900763;
stInitData.ModelParameters.param_robot.q_p_limit_upper[0] := 1.4835298641951802;
stInitData.ModelParameters.param_robot.q_p_limit_upper[1] := 1.4835298641951802;
stInitData.ModelParameters.param_robot.q_p_limit_upper[2] := 1.7453292519943295;
stInitData.ModelParameters.param_robot.q_p_limit_upper[3] := 1.3089969389957472;
stInitData.ModelParameters.param_robot.q_p_limit_upper[4] := 2.2689280275926285;
stInitData.ModelParameters.param_robot.q_p_limit_upper[5] := 2.3561944901923448;
stInitData.ModelParameters.param_robot.q_p_limit_upper[6] := 2.3561944901923448;
stInitData.ModelParameters.param_robot.q_p_limit_lower[0] := -1.4835298641951802;
stInitData.ModelParameters.param_robot.q_p_limit_lower[1] := -1.4835298641951802;
stInitData.ModelParameters.param_robot.q_p_limit_lower[2] := -1.7453292519943295;
stInitData.ModelParameters.param_robot.q_p_limit_lower[3] := -1.3089969389957472;
stInitData.ModelParameters.param_robot.q_p_limit_lower[4] := -2.2689280275926285;
stInitData.ModelParameters.param_robot.q_p_limit_lower[5] := -2.3561944901923448;
stInitData.ModelParameters.param_robot.q_p_limit_lower[6] := -2.3561944901923448;
stInitData.ModelParameters.timing.T_optitrack := 0.0040000000000000001;
stInitData.ModelParameters.timing.T_iiwa := 0.000125;
stInitData.ModelParameters.timing.T_optiTask := 5.0000000000000002e-05;
stInitData.ModelParameters.timing.cycle_time_ratio := 80;
stInitData.ModelParameters.filter_tau_T_1[0] := 0.00039788735772973834;
stInitData.ModelParameters.filter_tau_T_1[1] := 0.00039788735772973834;
stInitData.ModelParameters.filter_tau_T_1[2] := 0.00039788735772973834;
stInitData.ModelParameters.filter_tau_T_1[3] := 0.00039788735772973834;
stInitData.ModelParameters.filter_tau_T_1[4] := 0.0003183098861837907;
stInitData.ModelParameters.filter_tau_T_1[5] := 0.00015915494309189535;
stInitData.ModelParameters.filter_tau_T_1[6] := 0.00015915494309189535;
stInitData.ModelParameters.filter_tau_p_T_1[0] := 0.00039788735772973834;
stInitData.ModelParameters.filter_tau_p_T_1[1] := 0.00039788735772973834;
stInitData.ModelParameters.filter_tau_p_T_1[2] := 0.00039788735772973834;
stInitData.ModelParameters.filter_tau_p_T_1[3] := 0.00039788735772973834;
stInitData.ModelParameters.filter_tau_p_T_1[4] := 0.0003183098861837907;
stInitData.ModelParameters.filter_tau_p_T_1[5] := 0.00015915494309189535;
stInitData.ModelParameters.filter_tau_p_T_1[6] := 0.00015915494309189535;
stInitData.ModelParameters.filter_tau_p_slow_T_1[0] := 0.00079577471545947667;
stInitData.ModelParameters.filter_tau_p_slow_T_1[1] := 0.00079577471545947667;
stInitData.ModelParameters.filter_tau_p_slow_T_1[2] := 0.00079577471545947667;
stInitData.ModelParameters.filter_tau_p_slow_T_1[3] := 0.00079577471545947667;
stInitData.ModelParameters.filter_tau_p_slow_T_1[4] := 0.00079577471545947667;
stInitData.ModelParameters.filter_tau_p_slow_T_1[5] := 0.00079577471545947667;
stInitData.ModelParameters.filter_tau_p_slow_T_1[6] := 0.00079577471545947667;
stInitData.ModelParameters.filter_tau_slow_T_1[0] := 0.00079577471545947667;
stInitData.ModelParameters.filter_tau_slow_T_1[1] := 0.00079577471545947667;
stInitData.ModelParameters.filter_tau_slow_T_1[2] := 0.00079577471545947667;
stInitData.ModelParameters.filter_tau_slow_T_1[3] := 0.00079577471545947667;
stInitData.ModelParameters.filter_tau_slow_T_1[4] := 0.00079577471545947667;
stInitData.ModelParameters.filter_tau_slow_T_1[5] := 0.00079577471545947667;
stInitData.ModelParameters.filter_tau_slow_T_1[6] := 0.00079577471545947667;
stInitData.ModelParameters.filter_theta_p_T_1[0] := 0.00039788735772973834;
stInitData.ModelParameters.filter_theta_p_T_1[1] := 0.00039788735772973834;
stInitData.ModelParameters.filter_theta_p_T_1[2] := 0.00039788735772973834;
stInitData.ModelParameters.filter_theta_p_T_1[3] := 0.00039788735772973834;
stInitData.ModelParameters.filter_theta_p_T_1[4] := 0.0003183098861837907;
stInitData.ModelParameters.filter_theta_p_T_1[5] := 0.00015915494309189535;
stInitData.ModelParameters.filter_theta_p_T_1[6] := 0.00015915494309189535;
stInitData.ModelParameters.filter_theta_p_slow_T_1[0] := 0.00079577471545947667;
stInitData.ModelParameters.filter_theta_p_slow_T_1[1] := 0.00079577471545947667;
stInitData.ModelParameters.filter_theta_p_slow_T_1[2] := 0.00079577471545947667;
stInitData.ModelParameters.filter_theta_p_slow_T_1[3] := 0.00079577471545947667;
stInitData.ModelParameters.filter_theta_p_slow_T_1[4] := 0.00079577471545947667;
stInitData.ModelParameters.filter_theta_p_slow_T_1[5] := 0.00079577471545947667;
stInitData.ModelParameters.filter_theta_p_slow_T_1[6] := 0.00079577471545947667;
stInitData.ModelParameters.filter_theta_slow_T_1[0] := 0.00079577471545947667;
stInitData.ModelParameters.filter_theta_slow_T_1[1] := 0.00079577471545947667;
stInitData.ModelParameters.filter_theta_slow_T_1[2] := 0.00079577471545947667;
stInitData.ModelParameters.filter_theta_slow_T_1[3] := 0.00079577471545947667;
stInitData.ModelParameters.filter_theta_slow_T_1[4] := 0.00079577471545947667;
stInitData.ModelParameters.filter_theta_slow_T_1[5] := 0.00079577471545947667;
stInitData.ModelParameters.filter_theta_slow_T_1[6] := 0.00079577471545947667;
stInitData.ModelParameters.sensor_torque_offset[0] := 0.53000000000000003;
stInitData.ModelParameters.sensor_torque_offset[1] := -0.095000000000000001;
stInitData.ModelParameters.sensor_torque_offset[2] := -0.189;
stInitData.ModelParameters.sensor_torque_offset[3] := 0.070000000000000007;
stInitData.ModelParameters.sensor_torque_offset[4] := -0.058000000000000003;
stInitData.ModelParameters.sensor_torque_offset[5] := 0.0025000000000000001;
stInitData.ModelParameters.sensor_torque_offset[6] := -0.12;
stInitData.ModelParameters.tau_fm_hat_Y0 := 0;
stInitData.ModelParameters.L_Value[0] := 200;
stInitData.ModelParameters.L_Value[1] := 200;
stInitData.ModelParameters.L_Value[2] := 300;
stInitData.ModelParameters.L_Value[3] := 300;
stInitData.ModelParameters.L_Value[4] := 500;
stInitData.ModelParameters.L_Value[5] := 1000;
stInitData.ModelParameters.L_Value[6] := 1000;
stInitData.ModelParameters.use_theta_p_hat_Value := 0;
stInitData.ModelParameters.use_q_p_Value := 0;
stInitData.ModelParameters.subtract_model_Value := 0;
stInitData.ModelParameters.tau_c_plus_Value[0] := 0;
stInitData.ModelParameters.tau_c_plus_Value[1] := 0;
stInitData.ModelParameters.tau_c_plus_Value[2] := 0;
stInitData.ModelParameters.tau_c_plus_Value[3] := 0;
stInitData.ModelParameters.tau_c_plus_Value[4] := 0;
stInitData.ModelParameters.tau_c_plus_Value[5] := 0;
stInitData.ModelParameters.tau_c_plus_Value[6] := 0.20000000000000001;
stInitData.ModelParameters.tau_c_minus_Value[0] := 0;
stInitData.ModelParameters.tau_c_minus_Value[1] := 0;
stInitData.ModelParameters.tau_c_minus_Value[2] := 0;
stInitData.ModelParameters.tau_c_minus_Value[3] := 0;
stInitData.ModelParameters.tau_c_minus_Value[4] := 0;
stInitData.ModelParameters.tau_c_minus_Value[5] := 0;
stInitData.ModelParameters.tau_c_minus_Value[6] := 0.28000000000000003;
stInitData.ModelParameters.E_Value[0] := 0;
stInitData.ModelParameters.E_Value[1] := 0;
stInitData.ModelParameters.E_Value[2] := 0;
stInitData.ModelParameters.E_Value[3] := 0;
stInitData.ModelParameters.E_Value[4] := 0;
stInitData.ModelParameters.E_Value[5] := 0;
stInitData.ModelParameters.E_Value[6] := 120;
stInitData.ModelParameters.tau_v_Value[0] := 0;
stInitData.ModelParameters.tau_v_Value[1] := 0;
stInitData.ModelParameters.tau_v_Value[2] := 0;
stInitData.ModelParameters.tau_v_Value[3] := 0;
stInitData.ModelParameters.tau_v_Value[4] := 0;
stInitData.ModelParameters.tau_v_Value[5] := 0;
stInitData.ModelParameters.tau_v_Value[6] := 0.5;
stInitData.ModelParameters.Constant_Value[0] := 0;
stInitData.ModelParameters.Constant_Value[1] := 0;
stInitData.ModelParameters.Constant_Value[2] := 0;
stInitData.ModelParameters.Constant_Value[3] := 0;
stInitData.ModelParameters.Constant_Value[4] := 0;
stInitData.ModelParameters.Constant_Value[5] := 0;
stInitData.ModelParameters.Constant_Value[6] := 0;
stInitData.ModelParameters.tau_d_gravcomp_q_Y0 := 0;
stInitData.ModelParameters.GravitationcompensationK_D_Value := 1;
stInitData.ModelParameters.slope_factor_Value := 1;
stInitData.ModelParameters.tau_d_joint_ea_Y0 := 0;
stInitData.ModelParameters.JointbasedEALinearizationK_I_Value := 0;
stInitData.ModelParameters.JointbasedEALinearizationK_0_Value := 100;
stInitData.ModelParameters.JointbasedEALinearizationK_1_Value := 20;
stInitData.ModelParameters.UnitDelay_InitialCondition := 0;
stInitData.ModelParameters.Constant_Value_f := 0.050000000000000003;
stInitData.ModelParameters.Constant_Value_d[0] := 0;
stInitData.ModelParameters.Constant_Value_d[1] := 0;
stInitData.ModelParameters.Constant_Value_d[2] := 0;
stInitData.ModelParameters.Constant_Value_d[3] := 0;
stInitData.ModelParameters.Constant_Value_d[4] := 0;
stInitData.ModelParameters.Constant_Value_d[5] := 0;
stInitData.ModelParameters.Constant_Value_d[6] := 0;
stInitData.ModelParameters.FictionCompensationEnabled_Value := 1;
stInitData.ModelParameters.Constant22_Value := 1;
stInitData.ModelParameters.Constant4_Value := 1;
stInitData.ModelParameters.Constant7_Value := 1;
stInitData.ModelParameters.Constant8_Value := 1;
stInitData.ModelParameters.Constant9_Value := 1;
stInitData.ModelParameters.Constant10_Value := 1;
stInitData.ModelParameters.Constant23_Value := 1;
stInitData.ModelParameters.UnitDelay1_InitialCondition := 0;
stInitData.ModelParameters.ManualSwitch2_CurrentSetting := 1;
stInitData.ModelParameters.ManualSwitch4_CurrentSetting := 0;
stInitData.ContextInfoArr_0_TaskOidHdr.indexGroup := 0;
stInitData.ContextInfoArr_0_TaskOidHdr.indexOffset := 16#03002060;
stInitData.ContextInfoArr_0_TaskOidHdr.cbData := SIZEOF(stInitData.ContextInfoArr_0_TaskOid);
stInitData.ContextInfoArr_0_TaskPriorityHdr.indexGroup := 0;
stInitData.ContextInfoArr_0_TaskPriorityHdr.indexOffset := 16#03002070;
stInitData.ContextInfoArr_0_TaskPriorityHdr.cbData := SIZEOF(stInitData.ContextInfoArr_0_TaskPriority);
stInitData.ContextInfoArr_0_TaskCycleTimeNsHdr.indexGroup := 0;
stInitData.ContextInfoArr_0_TaskCycleTimeNsHdr.indexOffset := 16#03002080;
stInitData.ContextInfoArr_0_TaskCycleTimeNsHdr.cbData := SIZEOF(stInitData.ContextInfoArr_0_TaskCycleTimeNs);
stInitData.ContextInfoArr_0_TaskPortHdr.indexGroup := 0;
stInitData.ContextInfoArr_0_TaskPortHdr.indexOffset := 16#03002090;
stInitData.ContextInfoArr_0_TaskPortHdr.cbData := SIZEOF(stInitData.ContextInfoArr_0_TaskPort);
stInitData.ContextInfoArr_0_TaskSortOrderHdr.indexGroup := 0;
stInitData.ContextInfoArr_0_TaskSortOrderHdr.indexOffset := 16#030020b0;
stInitData.ContextInfoArr_0_TaskSortOrderHdr.cbData := SIZEOF(stInitData.ContextInfoArr_0_TaskSortOrder);
stInitData.Header.cbData := SIZEOF(stInitData)-SIZEOF(stInitData.Header);
stInitData.Header.uiElmCnt := 11;


// set pointer to InitData structure
SetInitDataInfo(ADR(stInitData));

// set DataArea information
SetDataAreaInfo(ADR(arrDataAreas),2);
arrDataAreas[1].nDataAreaId := 0;
arrDataAreas[1].nSize := SIZEOF(stInput);
arrDataAreas[1].pPlcVar := ADR(stInput);
arrDataAreas[1].pModuleProcImg := 0;
arrDataAreas[1].eDataAreaType := E_TcMatSimDataAreaType.InputDst;
arrDataAreas[2].nDataAreaId := 1;
arrDataAreas[2].nSize := SIZEOF(stOutput);
arrDataAreas[2].pPlcVar := ADR(stOutput);
arrDataAreas[2].pModuleProcImg := 0;
arrDataAreas[2].eDataAreaType := E_TcMatSimDataAreaType.OutputSrc;


// initialize basic interface pointers and return
FB_init := SUCCEEDED(Init(oid));
                  
                
END_METHOD

METHOD Execute : HRESULT
                  
IF (SUCCEEDED(hResult)) THEN
  hResult := VerifyParameters();
END_IF

// update DataArea information
SetDataAreaInfo(ADR(arrDataAreas),2);
arrDataAreas[1].nDataAreaId := 0;
arrDataAreas[1].nSize := SIZEOF(stInput);
arrDataAreas[1].pPlcVar := ADR(stInput);
arrDataAreas[1].pModuleProcImg := 0;
arrDataAreas[1].eDataAreaType := E_TcMatSimDataAreaType.InputDst;
arrDataAreas[2].nDataAreaId := 1;
arrDataAreas[2].nSize := SIZEOF(stOutput);
arrDataAreas[2].pPlcVar := ADR(stOutput);
arrDataAreas[2].pModuleProcImg := 0;
arrDataAreas[2].eDataAreaType := E_TcMatSimDataAreaType.OutputSrc;

	
// call base method
Execute := SUPER^.Execute();
                  
                
END_METHOD

{attribute 'object_name' := 'VerifyParameters'}
METHOD VerifyParameters : HRESULT
  VAR
    moduleCallByParam : TctModuleCallByType;
  END_VAR
                  
IF (bParametersVerified) THEN
  VerifyParameters := Tc2_System.E_HRESULTAdsErr.HRESULT_ADS_NOERROR;
ELSE
  VerifyParameters := GetObjPara(stInitData.CallByHdr.indexOffset,SIZEOF(moduleCallByParam),ADR(moduleCallByParam));
  
  // check the "CallBy" parameter to be set to "Module"
  IF (SUCCEEDED(VerifyParameters) AND (moduleCallByParam <> TctModuleCallByType.Module)) THEN
      VerifyParameters := Tc2_System.E_HRESULTAdsErr.INVALIDPARM;
  END_IF
  
  // set the parameters verified flag
  bParametersVerified := SUCCEEDED(VerifyParameters);
END_IF
                  
                
END_METHOD

PROPERTY InitData : ST_controller_ballcatcherInitData
GET
                    InitData := stInitData;
                  
END_GET
SET
                    stInitData := InitData;
                  
END_SET
END_PROPERTY
END_FUNCTION_BLOCK
